// TIA Portal project "Grundkurs Aufgabe 7 NEU" (V15.1)
// Vorlageprojekt für das Buch mit Zielsystem S7-1200

(* hardware
DEVICE "S7-1200-Station_1"  S7-1200 Station
   slot 0: "Baugruppenträger_0"  Rack  V1.0
   slot 1: "SPS"  CPU 1212C AC/DC/Rly  6ES7 212-1BE40-0XB0  V4.2
*)

// ===== PLC "SPS"  CPU 1212C AC/DC/Rly =====

VAR_GLOBAL   // PLC tag table "Eingänge und Ausgänge"
   "Taster_Start" AT %E0.0 : Bool;   // Taster "Start" Bedienpult (Schließer)
   "NotAus" AT %E0.2 : Bool;   // NotAus Bedienpult (Öffner)
   "Lichttaster_Ausschieber1" AT %E0.4 : Bool;   // Lichttaster vor Ausschieber 1 (Schließer)
   "Motor_Foerderband" AT %A0.2 : Bool;   // Motor Förderband vorwärts
   "Taster_Stop" AT %E0.1 : Bool;   // Taster "Stop" Bedienpult (Öffner)
   "Leuchte_Start" AT %A0.0 : Bool;   // Leuchte "Start" Bedienpult
   "Leuchte_Stop" AT %A0.1 : Bool;   // Leuchte "Stop" Bedienpult
   "Lichttaster_Einlauf" AT %E0.3 : Bool;   // Lichttaster im Einlauf des Förderbandes (Schließer)
   "Lichttaster_Ausschieber2" AT %E0.5 : Bool;   // Lichttaster vor Ausschieber 2 (Schließer)
   "Ausschieber1_zustellen" AT %A0.3 : Bool;   // Ausschieber 1 ausfahren Richtung Rampe
   "Ausschieber1_Band" AT %A0.4 : Bool;   // Förderband Ausschieber 1 vorwärts
   "Lichttaster_Ausschieber3" AT %E0.6 : Bool;   // Lichttaster vor Ausschieber 3 (Schließer)
   "Ausschieber2_zustellen" AT %A0.5 : Bool;   // Ausschieber 2 ausfahren Richtung Rampe
   "Ausschieber2_Band" AT %A0.6 : Bool;   // Förderband Ausschieber 2 vorwärts
   "Ausschieber3_zustellen" AT %A0.7 : Bool;   // Ausschieber 3 ausfahren Richtung Rampe
   "Ausschieber3_Band" AT %A1.0 : Bool;   // Förderband Ausschieber 3 vorwärts
END_VAR

VAR_GLOBAL   // PLC tag table "Merker"
   "Anlage_Start" AT %M1.0 : Bool;   // Anlage läuft
   "Foerderband_belegt" AT %M1.1 : Bool;   // Paket liegt auf Förderband
   "Hilfsmerker_FN" AT %M100.0 : Bool;   // Hilfsmerker für negative Flanke
   "Ausschieber1_ansteuern" AT %M1.2 : Bool;   // Erstes Paket -> Rampe 1 wird benutzt
   "Ausschieber2_ansteuern" AT %M1.3 : Bool;   // Zweites Paket -> Rampe 2 wird benutzt
   "Ausschieber3_ansteuern" AT %M1.4 : Bool;   // Drittes Paket -> Rampe 3 wird benutzt
END_VAR

// folder: System blocks/Program resources

DATA_BLOCK "Einschaltverz_Foerderer"   // DB1
{ S7_Optimized_Access := 'TRUE' }
AUTHOR : Simatic
FAMILY : IEC
NAME : IEC_TMR
VERSION : 1.0
// stored: InstanceOfName IEC_TIMER
"IEC_TIMER"
BEGIN
END_DATA_BLOCK

DATA_BLOCK "Einschaltverz_Paket_abtransportiert"   // DB2
{ S7_Optimized_Access := 'TRUE' }
AUTHOR : Simatic
FAMILY : IEC
NAME : IEC_TMR
VERSION : 1.0
// stored: InstanceOfName IEC_TIMER
"IEC_TIMER"
BEGIN
END_DATA_BLOCK

DATA_BLOCK "Zaehler_Ausschieber1"   // DB3
{ S7_Optimized_Access := 'TRUE' }
AUTHOR : Simatic
FAMILY : IEC
NAME : CNTR
VERSION : 1.0
// stored: InstanceOfName IEC_COUNTER
"IEC_COUNTER"
BEGIN
END_DATA_BLOCK

DATA_BLOCK "Zaehler_Ausschieber2"   // DB4
{ S7_Optimized_Access := 'TRUE' }
AUTHOR : Simatic
FAMILY : IEC
NAME : CNTR
VERSION : 1.0
// stored: InstanceOfName IEC_COUNTER
"IEC_COUNTER"
BEGIN
END_DATA_BLOCK

DATA_BLOCK "Zaehler_Ausschieber3"   // DB5
{ S7_Optimized_Access := 'TRUE' }
AUTHOR : Simatic
FAMILY : IEC
NAME : CNTR
VERSION : 1.0
// stored: InstanceOfName IEC_COUNTER
"IEC_COUNTER"
BEGIN
END_DATA_BLOCK

// folder: (top level)

FUNCTION "Kopplung_FactoryIO_mit_PLCSIM" : Void   // FC9000, SCL
{ S7_Optimized_Access := 'TRUE' }
VERSION : 0.1
   VAR_TEMP
      rdTimeReturn : Int;
      outputTime : DTL;
      SyncVal : Byte;
      forVal : Int;
      forVal_2 : Int;
      Value : Byte;
   END_VAR
   VAR CONSTANT
      CompVal : Byte := 16#34;
      Value_01 : Byte := 16#11;
      Value_01_DW : DWord := 16#A165_D992;
      Value_02_DW : DWord := 16#58BE_4401;
   END_VAR
BEGIN

   #Value:=PEEK(area := 16#82,
        dbNumber := 0,
        byteOffset := 511);
   #Value := #Value + 1;

   POKE(area := 16#82,
        dbNumber := 0,
        byteOffset := 511,
        value := #Value);

   POKE(area:=16#81,
        dbNumber:=0,
        byteOffset:=1016,
        value:=#Value_01_DW);
   POKE(area := 16#81,
        dbNumber := 0,
        byteOffset := 1020,
        value := #Value_02_DW);

   POKE(area := 16#81,
        dbNumber := 0,
        byteOffset := 511,
        value := B#16#00);

   FOR #forVal := 0 TO 120 DO
       FOR #forVal_2:=0 TO 10 DO
           #rdTimeReturn:=RD_SYS_T(#outputTime);
           #rdTimeReturn := WR_SYS_T(#outputTime);
           #rdTimeReturn := RD_SYS_T(#outputTime);
           #rdTimeReturn := WR_SYS_T(#outputTime);
       END_FOR;
       #SyncVal:= PEEK(area := 16#81,
                      dbNumber := 0,
                      byteOffset := 511);
       IF #SyncVal = #CompVal THEN
          GOTO M_1;
       END_IF;
   END_FOR;
   RETURN;

   M_1:
   POKE(area := 16#81,
        dbNumber := 0,
        byteOffset := 511,
        value := B#16#0);
END_FUNCTION

ORGANIZATION_BLOCK "Main"   // OB1, FBD, ProgramCycle
TITLE = "Main Program Sweep (Cycle)"
{ S7_Optimized_Access := 'TRUE' }
VERSION : 0.1
   VAR_INPUT
      Initial_Call : Bool;   // Initial call of this OB
      Remanence : Bool;   // =True, if remanent data are available
   END_VAR
BEGIN

REGION Network 1: Konnektierungsbaustein für PLC-Lab / Bausteinaufruf FC9000 (Für Aufgabe nicht relevant)
   // Im Netzwerk 1 wird der Konnektierungsbaustein für PLC-Lab aufgerufen.
   // Dieser Aufruf darf nicht entfernt werden!
   // Der Baustein FC9000 organisiert den Datentransfer zwischen PLCSIM und FactoryIO.
   // Der Baustein kann als Beispielprojekt von der FactoryIO-Homepage heruntergeladen werden.
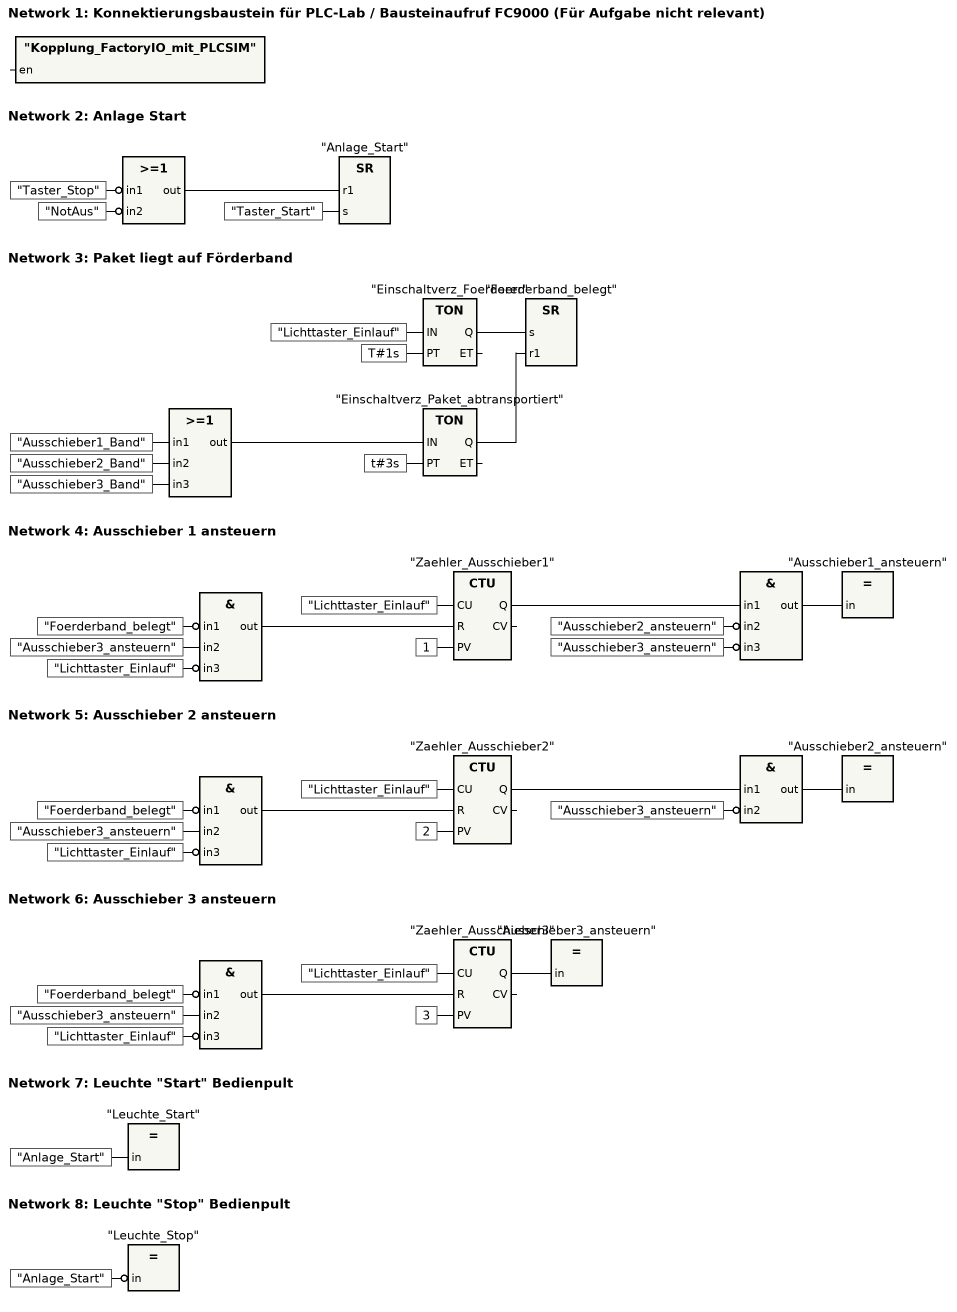
   "Kopplung_FactoryIO_mit_PLCSIM"();
END_REGION

REGION Network 2: Anlage Start
   IF "Taster_Start" THEN
       "Anlage_Start" := TRUE;   // SR flip-flop
   END_IF;
   IF NOT "Taster_Stop" OR NOT "NotAus" THEN "Anlage_Start" := FALSE; END_IF;
END_REGION

REGION Network 3: Paket liegt auf Förderband
   "Einschaltverz_Foerderer".TON(IN := "Lichttaster_Einlauf", PT := T#1s);
   "Einschaltverz_Paket_abtransportiert".TON(IN := "Ausschieber1_Band" OR "Ausschieber2_Band" OR "Ausschieber3_Band",
                           PT := t#3s);
   IF "Einschaltverz_Foerderer".Q THEN
       "Foerderband_belegt" := TRUE;   // SR flip-flop
   END_IF;
   IF "Einschaltverz_Paket_abtransportiert".Q THEN "Foerderband_belegt" := FALSE; END_IF;
END_REGION

REGION Network 4: Ausschieber 1 ansteuern
   "Zaehler_Ausschieber1".CTU(CU := "Lichttaster_Einlauf",
                           R := NOT "Foerderband_belegt" AND "Ausschieber3_ansteuern" AND NOT "Lichttaster_Einlauf",
                           PV := 1);
   "Ausschieber1_ansteuern" := "Zaehler_Ausschieber1".Q AND NOT "Ausschieber2_ansteuern" AND NOT "Ausschieber3_ansteuern";
END_REGION

REGION Network 5: Ausschieber 2 ansteuern
   "Zaehler_Ausschieber2".CTU(CU := "Lichttaster_Einlauf",
                           R := NOT "Foerderband_belegt" AND "Ausschieber3_ansteuern" AND NOT "Lichttaster_Einlauf",
                           PV := 2);
   "Ausschieber2_ansteuern" := "Zaehler_Ausschieber2".Q AND NOT "Ausschieber3_ansteuern";
END_REGION

REGION Network 6: Ausschieber 3 ansteuern
   "Zaehler_Ausschieber3".CTU(CU := "Lichttaster_Einlauf",
                           R := NOT "Foerderband_belegt" AND "Ausschieber3_ansteuern" AND NOT "Lichttaster_Einlauf",
                           PV := 3);
   "Ausschieber3_ansteuern" := "Zaehler_Ausschieber3".Q;
END_REGION

REGION Network 7: Leuchte "Start" Bedienpult
   "Leuchte_Start" := "Anlage_Start";
END_REGION

REGION Network 8: Leuchte "Stop" Bedienpult
   "Leuchte_Stop" := NOT "Anlage_Start";
END_REGION

REGION Network 9: Motor Förderband vorwärts
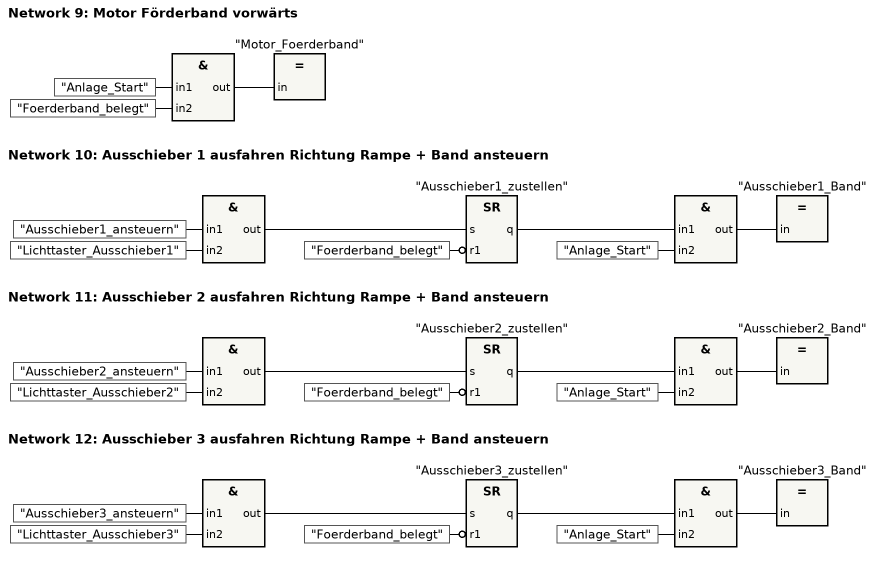
   "Motor_Foerderband" := "Anlage_Start" AND "Foerderband_belegt";
END_REGION

REGION Network 10: Ausschieber 1 ausfahren Richtung Rampe + Band ansteuern
   IF "Ausschieber1_ansteuern" AND "Lichttaster_Ausschieber1" THEN
       "Ausschieber1_zustellen" := TRUE;   // SR flip-flop
   END_IF;
   IF NOT "Foerderband_belegt" THEN "Ausschieber1_zustellen" := FALSE; END_IF;
   "Ausschieber1_Band" := "Ausschieber1_zustellen" AND "Anlage_Start";
END_REGION

REGION Network 11: Ausschieber 2 ausfahren Richtung Rampe + Band ansteuern
   IF "Ausschieber2_ansteuern" AND "Lichttaster_Ausschieber2" THEN
       "Ausschieber2_zustellen" := TRUE;   // SR flip-flop
   END_IF;
   IF NOT "Foerderband_belegt" THEN "Ausschieber2_zustellen" := FALSE; END_IF;
   "Ausschieber2_Band" := "Ausschieber2_zustellen" AND "Anlage_Start";
END_REGION

REGION Network 12: Ausschieber 3 ausfahren Richtung Rampe + Band ansteuern
   IF "Ausschieber3_ansteuern" AND "Lichttaster_Ausschieber3" THEN
       "Ausschieber3_zustellen" := TRUE;   // SR flip-flop
   END_IF;
   IF NOT "Foerderband_belegt" THEN "Ausschieber3_zustellen" := FALSE; END_IF;
   "Ausschieber3_Band" := "Ausschieber3_zustellen" AND "Anlage_Start";
END_REGION
END_ORGANIZATION_BLOCK